FUNCTION_BLOCK FB_AirHandlingUnit EXTENDS FB_ActuatorContinous
VAR_INPUT
END_VAR
VAR_OUTPUT
END_VAR
VAR

	localDefaultParameters : ST_AirHandlingUnitDefaultParameters;
	
	//analog converters
	OutputConverter : FB_AnalogOutput(fUpperLimit := 100, fLowerLimit := 0);
	
	//I/O Links
	bSetStatusOn_OUT	AT %Q* : BOOL;
	nSetPoint_OUT 		AT %Q* : INT;
	
END_VAR

MAIN();
OutputConverter(fValue := fSetPoint);

METHOD GetState : BOOL
VAR_INPUT
END_VAR
//local state
bStatusOn := controlState.bStatusOn;
END_METHOD

METHOD PROTECTED  SetSetPointLimits : BOOL
VAR_INPUT
END_VAR
aSetPointLimits[1] := 0;
aSetPointLimits[2] := 100;
END_METHOD

METHOD SetState : BOOL
VAR_INPUT
END_VAR
setPointState.fSetPoint := fSetPoint;
setPointState.aSetPointLimits := aSetPointLimits;
setPointState.sSetPointUnit := 'degreeC';

nSetPoint_OUT := OutputConverter.nValue;  //converts real setpoint for terminal
bSetStatusOn_OUT := NOT bSetStatusOn;		// must be inverted, because AHU is on, when do is 0
END_METHOD

END_FUNCTION_BLOCK

(* stored: Version 1.1.0.1, ProductVersion 3.1.4024.6
   POU FB_AirHandlingUnit: Id {f28cf46e-457c-4e41-bf4b-0887fb928971}, SpecialFunc None
   Method GetState: Id {db35ed20-518e-462b-86bf-ccce87aef9cc}
   Method SetSetPointLimits: Id {0bc4e5ec-6ce0-4801-843a-b7c2ee2178da}
   Method SetState: Id {524711c4-60d0-4e9d-aff4-c7e748d9a2be} *)
